FUNCTION_BLOCK ADP_HISTORY2 (* Offline identification prototype; see docs/adaptive/4diac-design.md *)
  (* Standard: 61499-2 *)
  (* Version 0.1, 2026-09-26, Guilherme *)
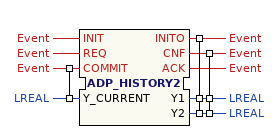
  EVENT_INPUT
    INIT;
    REQ;
    COMMIT WITH Y_CURRENT;
  END_EVENT
  EVENT_OUTPUT
    INITO WITH Y1, Y2;
    CNF WITH Y1, Y2;
    ACK;
  END_EVENT
  VAR_INPUT
    Y_CURRENT : LREAL;
  END_VAR
  VAR_OUTPUT
    Y1 : LREAL;
    Y2 : LREAL;
  END_VAR
  VAR
    H1 : LREAL;
    H2 : LREAL;
  END_VAR
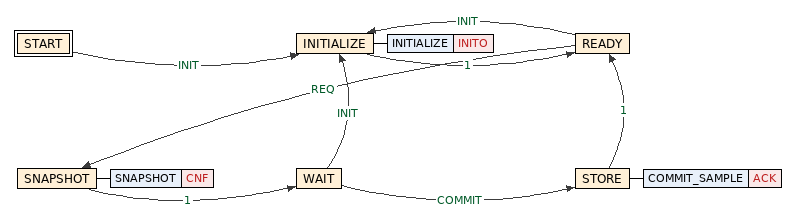
  EC_STATES
    START;
    INITIALIZE : INITIALIZE -> INITO;
    READY;
    SNAPSHOT : SNAPSHOT -> CNF;
    WAIT;
    STORE : COMMIT_SAMPLE -> ACK;
  END_STATES
  EC_TRANSITIONS
    START TO INITIALIZE := INIT;
    INITIALIZE TO READY := 1;
    READY TO INITIALIZE := INIT;
    READY TO SNAPSHOT := REQ;
    SNAPSHOT TO WAIT := 1;
    WAIT TO INITIALIZE := INIT;
    WAIT TO STORE := COMMIT;
    STORE TO READY := 1;
  END_TRANSITIONS
  ALGORITHM INITIALIZE IN ST:
H1 := 0.0;
H2 := 0.0;
Y1 := 0.0;
Y2 := 0.0;
  END_ALGORITHM
  ALGORITHM SNAPSHOT IN ST:
Y1 := H1;
Y2 := H2;
  END_ALGORITHM
  ALGORITHM COMMIT_SAMPLE IN ST:
H2 := H1;
H1 := Y_CURRENT;
  END_ALGORITHM
END_FUNCTION_BLOCK
